FUNCTION TryConvert_UINT_TO_TOD : BOOL
VAR_INPUT
	in : UINT;
	out : REFERENCE TO TOD;
END_VAR

out := UINT_TO_TOD(in);
TryConvert_UINT_TO_TOD := TRUE;

END_FUNCTION

(* stored: Version 1.1.0.1, ProductVersion 3.1.4024.12
   POU TryConvert_UINT_TO_TOD: Id {8cc03be3-7b32-4ce3-89b3-5717a2d912cb}, SpecialFunc None *)
